FUNCTION_BLOCK FB_Convert_2temp
VAR_INPUT
	iInput			:	INT;
	tRefresh		:	TIME;
	itempMAX		:	INT;
	iTempMIN		:	INT;
END_VAR
VAR_OUTPUT
	wOut			:	WORD;
END_VAR
VAR
	rX				:	REAL;
	tonBlock		:	TON;
	
	rMaxTempStep	:	REAL;
	rValuePerStep	:	REAL;
	bInit			:	BOOL := FALSE;
	iOut			:	INT;
END_VAR

// For Convertion of 0-10V Signal from 0-100%
tonBlock(IN := NOT tonBlock.Q, PT := tRefresh);

IF NOT bInit THEN
	rMaxTempStep	:= INT_TO_REAL(iTempMax + (iTempMin * (-1)));
	rValuePerStep	:= (rMaxTempStep / INT_TO_REAL(32767));

	bInit := TRUE;
END_IF


IF tonBlock.Q THEN

	rX := INT_TO_REAL(iInput) * rValuePerStep;
	
	rX := rX + INT_TO_REAL(iTempMIN);

	
	iOut := REAL_TO_INT(rX * 10.0);
	wOut := INT_TO_WORD(iOut);
	
END_IF

END_FUNCTION_BLOCK

(* stored: Version 1.1.0.1, ProductVersion 3.1.4024.13
   POU FB_Convert_2temp: Id {1aef795d-fbd2-4a71-be44-896f67cfdb69}, SpecialFunc None *)
